// TIA Portal V20 export
FUNCTION "LER_PartData_VisionTriggerPos" : Void   // FC10002, LAD
// stored: Access Published, SetENOAutomatically false
   VAR_INPUT
      generateCondition : Bool;
      specialFunctions : "LAF_typeSpecialFunctions";
      recipeNo : Int;
      processUnitSelect : Int;   // 1. Anode Reel Cut, 2. Cathode Reel Cut, 3. Stacking#1, 4.Stacking#2, 5. Inspection
      bobinID : String;
   END_VAR
   VAR_OUTPUT
      PartData : "LER_typePartData";
   END_VAR
   VAR_TEMP
      tempRET_VAL : Word;
   END_VAR
   VAR CONSTANT
      PartStatus_PartsAvailable : Byte := 16#1;
      AnodeMachineNumber : Byte := 16#A;
      CathodeMachineNumber : Byte := 16#F;
   END_VAR
BEGIN

REGION Network 1: PartType
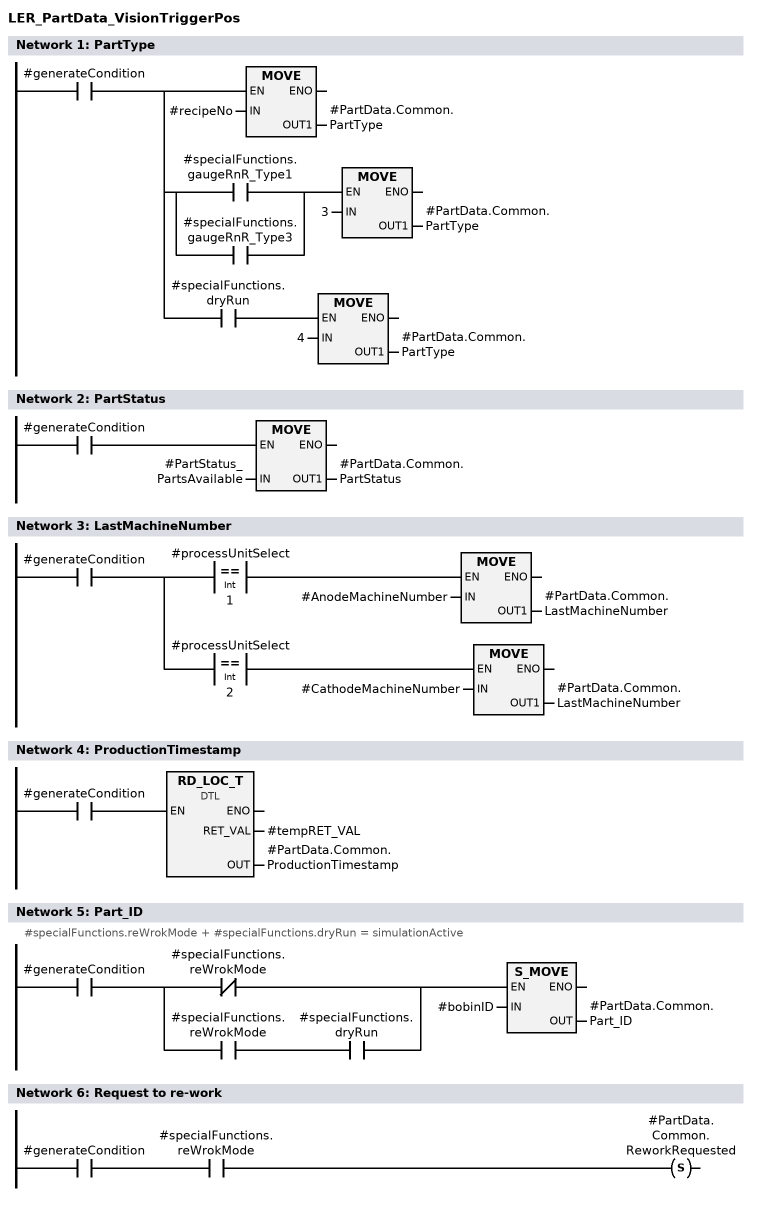
   RUNG wire#powerrail
      Contact( #generateCondition )
      wire#w1
      Move(in := #recipeNo, out1 => #PartData.Common.PartType)
   END_RUNG
   RUNG wire#w1
      Contact( #specialFunctions.gaugeRnR_Type1 )
      wire#w2
      Move(in := 3, out1 => #PartData.Common.PartType)
   END_RUNG
   RUNG wire#w1
      Contact( #specialFunctions.gaugeRnR_Type3 )
   END_RUNG wire#w2
   RUNG wire#w1
      Contact( #specialFunctions.dryRun )
      Move(in := 4, out1 => #PartData.Common.PartType)
   END_RUNG
   // the same network as SCL:
   IF #generateCondition THEN #PartData.Common.PartType := #recipeNo; END_IF;
   IF #generateCondition AND (#specialFunctions.gaugeRnR_Type1 OR #specialFunctions.gaugeRnR_Type3) THEN
       #PartData.Common.PartType := 3;
   END_IF;
   IF #generateCondition AND #specialFunctions.dryRun THEN #PartData.Common.PartType := 4; END_IF;
END_REGION

REGION Network 2: PartStatus
   RUNG wire#powerrail
      Contact( #generateCondition )
      Move(in := #PartStatus_PartsAvailable, out1 => #PartData.Common.PartStatus)
   END_RUNG
   // the same network as SCL:
   IF #generateCondition THEN #PartData.Common.PartStatus := #PartStatus_PartsAvailable; END_IF;
END_REGION

REGION Network 3: LastMachineNumber
   RUNG wire#powerrail
      Contact( #generateCondition )
      wire#w1
      { S7_Templates := "SrcType := Int" } EQ_Contact(in1 := #processUnitSelect, in2 := 1)
      Move(in := #AnodeMachineNumber, out1 => #PartData.Common.LastMachineNumber)
   END_RUNG
   RUNG wire#w1
      { S7_Templates := "SrcType := Int" } EQ_Contact(in1 := #processUnitSelect, in2 := 2)
      Move(in := #CathodeMachineNumber, out1 => #PartData.Common.LastMachineNumber)
   END_RUNG
   // the same network as SCL:
   IF #generateCondition AND (#processUnitSelect = 1) THEN
       #PartData.Common.LastMachineNumber := #AnodeMachineNumber;
   END_IF;
   IF #generateCondition AND (#processUnitSelect = 2) THEN
       #PartData.Common.LastMachineNumber := #CathodeMachineNumber;
   END_IF;
END_REGION

REGION Network 4: ProductionTimestamp
   RUNG wire#powerrail
      Contact( #generateCondition )
      { S7_Templates := "date_type := DTL" } RD_LOC_T(RET_VAL => #tempRET_VAL, OUT => #PartData.Common.ProductionTimestamp)
   END_RUNG
   // the same network as SCL:
   IF #generateCondition THEN #tempRET_VAL := RD_LOC_T(OUT => #PartData.Common.ProductionTimestamp); END_IF;
END_REGION

REGION Network 5: Part_ID
   // #specialFunctions.reWrokMode + #specialFunctions.dryRun = simulationActive
   RUNG wire#powerrail
      Contact( #generateCondition )
      wire#w1
      I_Contact( #specialFunctions.reWrokMode )
      wire#w2
      S_Move(in := #bobinID, out => #PartData.Common.Part_ID)
   END_RUNG
   RUNG wire#w1
      Contact( #specialFunctions.reWrokMode )
      Contact( #specialFunctions.dryRun )
   END_RUNG wire#w2
   // the same network as SCL:
   IF #generateCondition AND (NOT #specialFunctions.reWrokMode OR (#specialFunctions.reWrokMode AND #specialFunctions.dryRun)) THEN
       #PartData.Common.Part_ID := #bobinID;
   END_IF;
END_REGION

REGION Network 6: Request to re-work
   RUNG wire#powerrail
      Contact( #generateCondition )
      Contact( #specialFunctions.reWrokMode )
      S_Coil( #PartData.Common.ReworkRequested )
   END_RUNG
   // the same network as SCL:
   IF #generateCondition AND #specialFunctions.reWrokMode THEN
       #PartData.Common.ReworkRequested := TRUE;
   END_IF;
END_REGION
END_FUNCTION
